// Mitsubishi GX Works2 project: servo_motor_ex8_block-loop   PLC: Q02/Q02H

PROGRAM MAIN
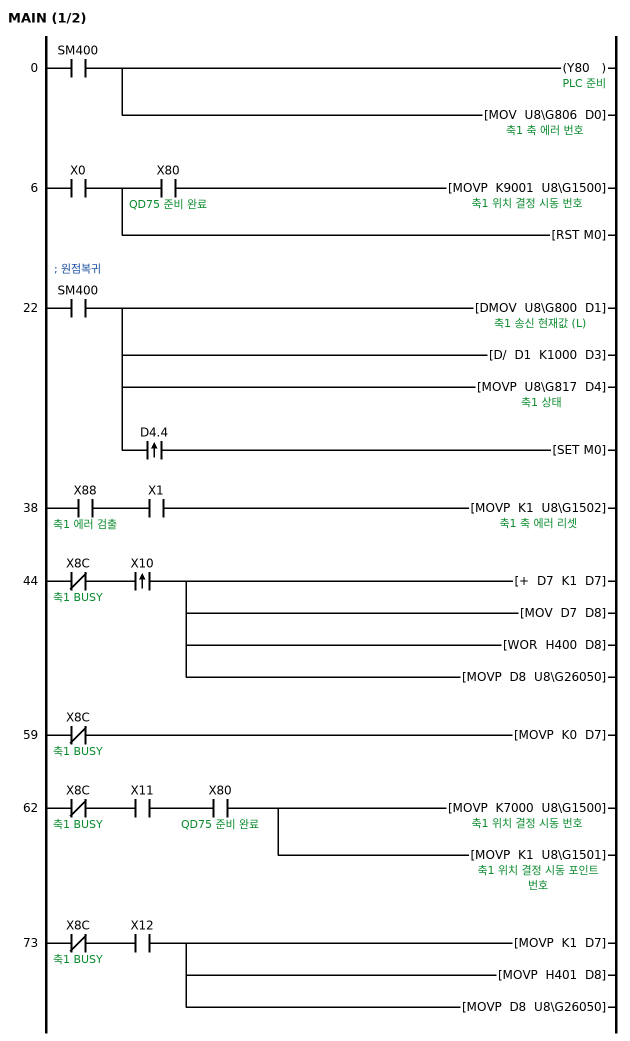
0     LD      SM400
      OUT     Y80  ; PLC 준비
      MOV     U8\G806 D0  ; 축1 축 에러 번호
6     LD      X0
      MPS
      AND     X80  ; QD75 준비 완료
      MOVP    K9001 U8\G1500  ; 축1 위치 결정 시동 번호
      MPP
      RST     M0
; 원점복귀
22    LD      SM400
      DMOV    U8\G800 D1  ; 축1 송신 현재값 (L)
      D/      D1 K1000 D3
      MOVP    U8\G817 D4  ; 축1 상태
      ANDP    D4.4
      SET     M0
38    LD      X88  ; 축1 에러 검출
      AND     X1
      MOVP    K1 U8\G1502  ; 축1 축 에러 리셋
44    LDI     X8C  ; 축1 BUSY
      ANDP    X10
      +       D7 K1 D7
      MOV     D7 D8
      WOR     H400 D8
      MOVP    D8 U8\G26050
59    LDI     X8C  ; 축1 BUSY
      MOVP    K0 D7
62    LDI     X8C  ; 축1 BUSY
      AND     X11
      AND     X80  ; QD75 준비 완료
      MOVP    K7000 U8\G1500
      MOVP    K1 U8\G1501  ; 축1 위치 결정 시동 포인트 번호
73    LDI     X8C  ; 축1 BUSY
      AND     X12
      MOVP    K1 D7
      MOVP    H401 D8
      MOVP    D8 U8\G26050
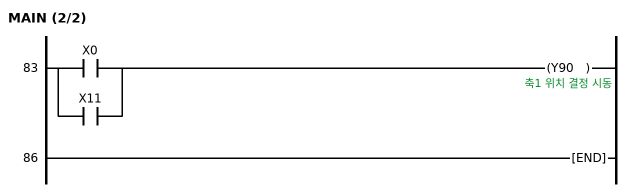
83    LD      X0
      OR      X11
      OUT     Y90  ; 축1 위치 결정 시동
86    END
END_PROGRAM

// device comments not shown above
X81  ; 동기용 플래그
X84  ; 축1 M 코드 ON
X85  ; 축2 M 코드 ON
X89  ; 축2 에러 검출
X8D  ; 축2 BUSY
X90  ; 축1 시동 완료
X91  ; 축2 시동 완료
X94  ; 축1 위치 결정 완료
X95  ; 축2 위치 결정 완료
Y84  ; 축1 축 정지
Y85  ; 축2 축 정지
Y88  ; 축1 정운전 JOG 시동
Y89  ; 축1 역운전 JOG 시동
Y8A  ; 축2 정운전 JOG 시동
Y8B  ; 축2 역운전 JOG 시동
Y91  ; 축2 위치 결정 시동
Y94  ; 축1 실행 금지 플래그
Y95  ; 축2 실행 금지 플래그
